TYPE STMInfoData :
STRUCT
	infoData1 : UINT;
	infoData2 : UINT;
	infoData3 : UINT;
END_STRUCT
END_TYPE

(* stored: Version 1.1.0.1, ProductVersion 3.1.4024.9
   DUT STMInfoData: Id {1d6f213d-8665-415c-ae1c-d6f8ff2600bb} *)
